// TIA Portal V19 export
VAR_GLOBAL   // PLC tag table "00_Simulation"
END_VAR
